RoboDK station: Station Basic Pick Box.rdk

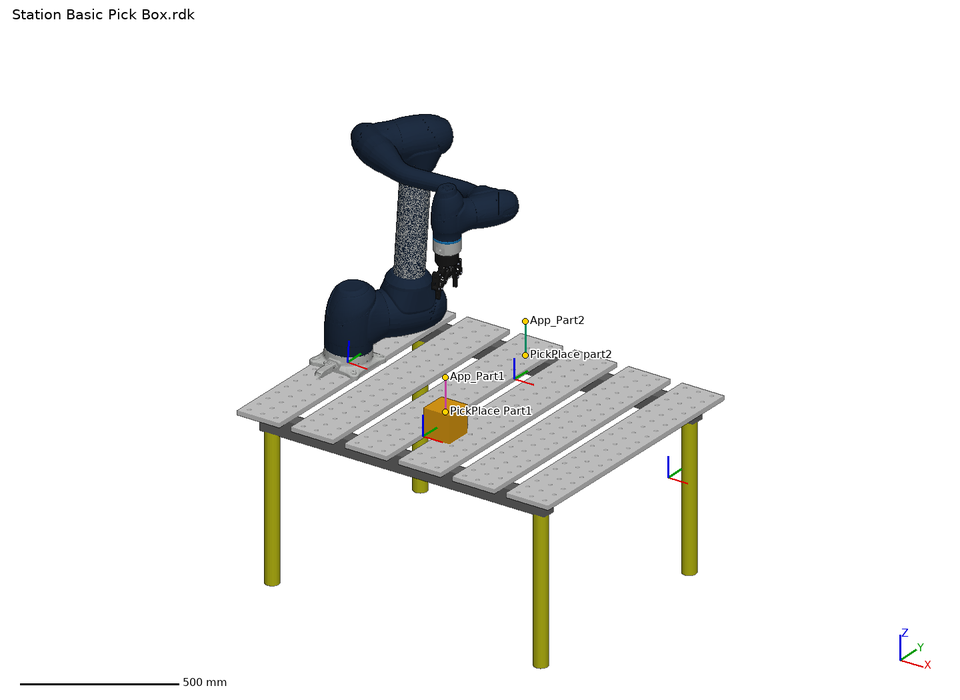
[picture v0: the station drawn from its stored meshes, robots at their saved joint values, targets as dots, program paths as lines]
Station Station Basic Pick Box (saved by RoboDK 6.0.5). Poses are relative to the parent item; angles as X-Y-Z fixed-axis rotations.
  - frame Doosan Robotics M1013 Base at (-800, 100, 0) mm, rotated rx 0 ry 3.23 rz 0 deg
    - robot Doosan Robotics M1013: 6 axes, payload 10 kg, reach 1300 mm, repeatability 0.05 mm, weight 33 kg
        modified DH rows (alpha deg, a mm, theta deg, d mm): 0, 0, 0, 152.5; -90, 0, -90, -34.506; 0, 620, -90, 0; -90, 0, 0, 559; 90, 0, 0, 0; -90, 0, 180, 121
        base shift (0, 0, 0) mm, rotated rx 0 ry 0 rz 180 deg
        joint limits [-360, -360, -160, -360, -360, -360] to [360, 360, 160, 360, 360, 360]; home [0, 0, 90, 0, 0, 0]; saved at [-29.41, 1.078, 86.928, 1.206, 89.854, 56.633]
      - tool RobotiQ 2F-85 Gripper (Open), TCP at (0, 0, 130) mm, size 147.4 x 75 x 146.8 mm
  - frame World at (500, 0, 0) mm
    - object Table 1200x1000mm (Welding) at (-790, 100, 0) mm, size 1193.8 x 965.2 x 609.6 mm, geometry from Table-1200x1000mm-Welding.sld
  - frame Part1 at (-300, -200, 0) mm
    - target PickPlace Part1 (Cartesian target) at (50, 50, 80) mm, rotated rx -179.22 ry -0.05 rz 93.98 deg; joints [-28.449, 17.055, 116.272, 1.668, 44.525, 56.407] of Doosan Robotics M1013
    - target App_Part1 (Cartesian target) at (50, 50, 200) mm, rotated rx -179.22 ry -0.05 rz 93.98 deg; joints [-28.766, 9.3, 111.099, 1.402, 57.455, 56.525] of Doosan Robotics M1013
    - target Target 3 (Cartesian target) at (50, 50, 200) mm, rotated rx -179.22 ry -0.05 rz 93.98 deg; joints [-28.766, 9.3, 111.099, 1.402, 57.455, 56.525] of Doosan Robotics M1013
    - target Target 4 (Cartesian target) at (50, 50, 200) mm, rotated rx -179.22 ry -0.05 rz 93.98 deg; joints [-28.766, 9.3, 111.099, 1.402, 57.455, 56.525] of Doosan Robotics M1013
    - object Box at (0, 0, 0) mm, size 100 x 100 x 100 mm, geometry from Cube-100mm.sld
  - program ReplaceObjects (1 instructions, listed below)
  - program PickPart1 (6 instructions, listed below)
  - frame Part2 at (-300, 300, 0) mm
    - target App_Part2 (Cartesian target) at (25, 25, 200) mm, rotated rx -179.22 ry -0.05 rz 93.98 deg; joints [20.542, 6.511, 114.552, -1.032, 56.641, 107.116] of Doosan Robotics M1013
    - target PickPlace part2 (Cartesian target) at (25, 25, 80) mm, rotated rx -179.22 ry -0.05 rz 93.98 deg; joints [20.296, 14.657, 119.879, -1.245, 43.167, 107.212] of Doosan Robotics M1013
  - program PlacePart2 (6 instructions, listed below)
  - program PickPart2 (6 instructions, listed below)
  - program PlacePart1 (6 instructions, listed below)
  - program Programme Principal (4 instructions, listed below)
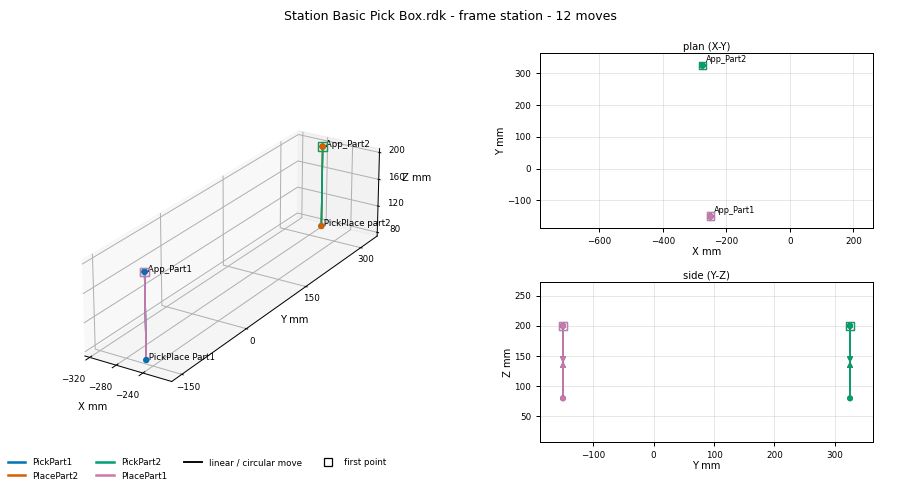
[picture p0: tool path of Station Basic Pick Box.rdk in frame station, 12 of 12 moves have a stored position in this frame; points joined in program order, loops and branches not executed]

--- program ReplaceObjects (robot Doosan Robotics M1013) ---
  Déplacer Box

--- program PickPart1 (robot Doosan Robotics M1013) ---
  Définir Ref.: Part1
  Choisir Outil: RobotiQ 2F-85 Gripper (Open)
  MoveJ (App_Part1)
  MoveL (PickPlace 1) -> target PickPlace Part1
  Attacher à RobotiQ 2F-85 Gripper (Open)
  MoveL (App_Part1)

--- program PlacePart2 (robot Doosan Robotics M1013) ---
  Définir Ref.: Part2
  Choisir Outil: RobotiQ 2F-85 Gripper (Open)
  MoveJ (App_Part2)
  MoveL (PickPlace part2)
  Détachez de RobotiQ 2F-85 Gripper (Open)
  MoveL (App_Part2)

--- program PickPart2 (robot Doosan Robotics M1013) ---
  Définir Ref.: Part2
  Choisir Outil: RobotiQ 2F-85 Gripper (Open)
  MoveJ (App_Part2)
  MoveL (PickPlace part2)
  Attacher à RobotiQ 2F-85 Gripper (Open)
  MoveL (App_Part2)

--- program PlacePart1 (robot Doosan Robotics M1013) ---
  Définir Ref.: Part1
  Choisir Outil: RobotiQ 2F-85 Gripper (Open)
  MoveJ (App_Part1)
  MoveL (PickPlace Part1)
  Détachez de RobotiQ 2F-85 Gripper (Open)
  MoveL (App_Part1)

--- program Programme Principal (robot Doosan Robotics M1013) ---
  Appel PickPart1
  Appel PlacePart2
  Appel PickPart2
  Appel PlacePart1
